{attribute 'GeneratedUsingTerminal: EL5072-0000-0016'}
{attribute addProperty BoxType "EL5072-0000-0016"}
{attribute addProperty Id "IND_Inputs_Channel_1AT %I*IND_Inputs_Channel_BBE8401F18IND_Inputs_Channel_2AT %I*IND_Inputs_Channel_BBE8401F18IND_Outputs_Channel_1AT %Q*IND_Outputs_Channel_02FDE6C97IND_Outputs_Channel_2AT %Q*IND_Outputs_Channel_02FDE6C97WcStateAT %I*WcState_9091E0EB2InfoDataAT %I*InfoData_94A18F5E2"}
{attribute addProperty CRC "3282016868"}
{attribute addProperty Size "54"}
TYPE EL5072_C39F9A64 EXTENDS EtcSlaveTerminalBase_947E5A46 :
STRUCT
	{attribute addProperty Name "IND_Inputs_Channel_1"}
	IND_Inputs_Channel_1 : IND_Inputs_Channel_BBE8401F;
	{attribute addProperty Name "IND_Inputs_Channel_2"}
	IND_Inputs_Channel_2 : IND_Inputs_Channel_BBE8401F;
	{attribute addProperty Name "IND_Outputs_Channel_1"}
	IND_Outputs_Channel_1 : IND_Outputs_Channel_02FDE6C9;
	{attribute addProperty Name "IND_Outputs_Channel_2"}
	IND_Outputs_Channel_2 : IND_Outputs_Channel_02FDE6C9;
	{attribute addProperty Name "WcState"}
	WcState : WcState_9091E0EB;
	{attribute addProperty Name "InfoData"}
	InfoData : InfoData_94A18F5E;
END_STRUCT
END_TYPE

(* stored: Version 1.2.0.0, ProductVersion 3.1.4024.9
   DUT EL5072_C39F9A64: Id {1333a5bd-3d39-4ad0-ac61-f7c3c68ddf3e} *)
